	X =  351.615  mm,	Y =   -114.701  mm,	Z =   -236.484  mm,
	W =  90.000 deg,	P =   0.000 deg,	R =   90.000 deg
};
P[3234]{
   GP1:
	UF : 0, UT : 6,		CONFIG : 'N U T, 0, 0, 0',
	X =  350.642  mm,	Y =   -113.945  mm,	Z =   -236.457  mm,
	W =  90.000 deg,	P =   0.000 deg,	R =   90.000 deg
};
P[3235]{
   GP1:
	UF : 0, UT : 6,		CONFIG : 'N U T, 0, 0, 0',
	X =  349.632  mm,	Y =   -113.307  mm,	Z =   -236.452  mm,
	W =  90.000 deg,	P =   0.000 deg,	R =   90.000 deg
};
P[3236]{
   GP1:
	UF : 0, UT : 6,		CONFIG : 'N U T, 0, 0, 0',
	X =  344.937  mm,	Y =   -111.604  mm,	Z =   -236.287  mm,
	W =  90.000 deg,	P =   0.000 deg,	R =   90.000 deg
};
P[3237]{
   GP1:
	UF : 0, UT : 6,		CONFIG : 'N U T, 0, 0, 0',
	X =  342.838  mm,	Y =   -111.355  mm,	Z =   -236.028  mm,
	W =  90.000 deg,	P =   0.000 deg,	R =   90.000 deg
};
P[3238]{
   GP1:
	UF : 0, UT : 6,		CONFIG : 'N U T, 0, 0, 0',
	X =  340.930  mm,	Y =   -111.626  mm,	Z =   -236.285  mm,
	W =  90.000 deg,	P =   0.000 deg,	R =   90.000 deg
};
P[3239]{
   GP1:
	UF : 0, UT : 6,		CONFIG : 'N U T, 0, 0, 0',
	X =  338.780  mm,	Y =   -112.047  mm,	Z =   -236.080  mm,
	W =  90.000 deg,	P =   0.000 deg,	R =   90.000 deg
};
P[3240]{
   GP1:
	UF : 0, UT : 6,		CONFIG : 'N U T, 0, 0, 0',
	X =  338.192  mm,	Y =   -112.362  mm,	Z =   -236.275  mm,
	W =  90.000 deg,	P =   0.000 deg,	R =   90.000 deg
};
P[3241]{
   GP1:
	UF : 0, UT : 6,		CONFIG : 'N U T, 0, 0, 0',
	X =  337.107  mm,	Y =   -112.912  mm,	Z =   -236.405  mm,
	W =  90.000 deg,	P =   0.000 deg,	R =   90.000 deg
};
P[3242]{
   GP1:
	UF : 0, UT : 6,		CONFIG : 'N U T, 0, 0, 0',
	X =  334.503  mm,	Y =   -114.254  mm,	Z =   -236.336  mm,
	W =  90.000 deg,	P =   0.000 deg,	R =   90.000 deg
};
P[3243]{
   GP1:
	UF : 0, UT : 6,		CONFIG : 'N U T, 0, 0, 0',
	X =  331.830  mm,	Y =   -115.833  mm,	Z =   -236.422  mm,
	W =  90.000 deg,	P =   0.000 deg,	R =   90.000 deg
};
P[3244]{
   GP1:
	UF : 0, UT : 6,		CONFIG : 'N U T, 0, 0, 0',
	X =  330.177  mm,	Y =   -116.811  mm,	Z =   -236.480  mm,
	W =  90.000 deg,	P =   0.000 deg,	R =   90.000 deg
};
P[3245]{
   GP1:
	UF : 0, UT : 6,		CONFIG : 'N U T, 0, 0, 0',
	X =  327.562  mm,	Y =   -118.180  mm,	Z =   -236.136  mm,
	W =  90.000 deg,	P =   0.000 deg,	R =   90.000 deg
};
P[3246]{
   GP1:
	UF : 0, UT : 6,		CONFIG : 'N U T, 0, 0, 0',
	X =  322.354  mm,	Y =   -121.298  mm,	Z =   -236.409  mm,
	W =  90.000 deg,	P =   0.000 deg,	R =   90.000 deg
};
P[3247]{
   GP1:
	UF : 0, UT : 6,		CONFIG : 'N U T, 0, 0, 0',
	X =  321.571  mm,	Y =   -121.625  mm,	Z =   -236.103  mm,
	W =  90.000 deg,	P =   0.000 deg,	R =   90.000 deg
};
P[3248]{
   GP1:
	UF : 0, UT : 6,		CONFIG : 'N U T, 0, 0, 0',
	X =  320.626  mm,	Y =   -122.310  mm,	Z =   -236.441  mm,
	W =  90.000 deg,	P =   0.000 deg,	R =   90.000 deg
};
P[3249]{
   GP1:
	UF : 0, UT : 6,		CONFIG : 'N U T, 0, 0, 0',
	X =  319.747  mm,	Y =   -122.679  mm,	Z =   -236.108  mm,
	W =  90.000 deg,	P =   0.000 deg,	R =   90.000 deg
};
P[3250]{
   GP1:
	UF : 0, UT : 6,		CONFIG : 'N U T, 0, 0, 0',
	X =  317.760  mm,	Y =   -123.868  mm,	Z =   -236.208  mm,
	W =  90.000 deg,	P =   0.000 deg,	R =   90.000 deg
};
P[3251]{
   GP1:
	UF : 0, UT : 6,		CONFIG : 'N U T, 0, 0, 0',
	X =  317.024  mm,	Y =   -124.291  mm,	Z =   -236.201  mm,
	W =  90.000 deg,	P =   0.000 deg,	R =   90.000 deg
};
P[3252]{
   GP1:
	UF : 0, UT : 6,		CONFIG : 'N U T, 0, 0, 0',
	X =  311.457  mm,	Y =   -127.567  mm,	Z =   -236.352  mm,
	W =  90.000 deg,	P =   0.000 deg,	R =   90.000 deg
};
P[3253]{
   GP1:
	UF : 0, UT : 6,		CONFIG : 'N U T, 0, 0, 0',
	X =  308.513  mm,	Y =   -129.171  mm,	Z =   -236.117  mm,
	W =  90.000 deg,	P =   0.000 deg,	R =   90.000 deg
};
P[3254]{
   GP1:
	UF : 0, UT : 6,		CONFIG : 'N U T, 0, 0, 0',
	X =  303.378  mm,	Y =   -132.275  mm,	Z =   -236.456  mm,
	W =  90.000 deg,	P =   0.000 deg,	R =   90.000 deg
};
P[3255]{
   GP1:
	UF : 0, UT : 6,		CONFIG : 'N U T, 0, 0, 0',
	X =  302.185  mm,	Y =   -132.859  mm,	Z =   -236.203  mm,
	W =  90.000 deg,	P =   0.000 deg,	R =   90.000 deg
};
P[3256]{
   GP1:
	UF : 0, UT : 6,		CONFIG : 'N U T, 0, 0, 0',
	X =  301.114  mm,	Y =   -133.543  mm,	Z =   -236.361  mm,
	W =  90.000 deg,	P =   0.000 deg,	R =   90.000 deg
};
P[3257]{
   GP1:
	UF : 0, UT : 6,		CONFIG : 'N U T, 0, 0, 0',
	X =  299.155  mm,	Y =   -134.553  mm,	Z =   -236.068  mm,
	W =  90.000 deg,	P =   0.000 deg,	R =   90.000 deg
};
P[3258]{
   GP1:
	UF : 0, UT : 6,		CONFIG : 'N U T, 0, 0, 0',
	X =  298.148  mm,	Y =   -135.225  mm,	Z =   -236.288  mm,
	W =  90.000 deg,	P =   0.000 deg,	R =   90.000 deg
};
P[3259]{
   GP1:
	UF : 0, UT : 6,		CONFIG : 'N U T, 0, 0, 0',
	X =  295.503  mm,	Y =   -136.793  mm,	Z =   -236.386  mm,
	W =  90.000 deg,	P =   0.000 deg,	R =   90.000 deg
};
P[3260]{
   GP1:
	UF : 0, UT : 6,		CONFIG : 'N U T, 0, 0, 0',
	X =  294.548  mm,	Y =   -137.306  mm,	Z =   -236.294  mm,
	W =  90.000 deg,	P =   0.000 deg,	R =   90.000 deg
};
P[3261]{
   GP1:
	UF : 0, UT : 6,		CONFIG : 'N U T, 0, 0, 0',
	X =  291.446  mm,	Y =   -139.089  mm,	Z =   -236.273  mm,
	W =  90.000 deg,	P =   0.000 deg,	R =   90.000 deg
};
P[3262]{
   GP1:
	UF : 0, UT : 6,		CONFIG : 'N U T, 0, 0, 0',
	X =  288.476  mm,	Y =   -140.784  mm,	Z =   -236.224  mm,
	W =  90.000 deg,	P =   0.000 deg,	R =   90.000 deg
};
P[3263]{
   GP1:
	UF : 0, UT : 6,		CONFIG : 'N U T, 0, 0, 0',
	X =  287.259  mm,	Y =   -141.421  mm,	Z =   -236.065  mm,
	W =  90.000 deg,	P =   0.000 deg,	R =   90.000 deg
};
P[3264]{
   GP1:
	UF : 0, UT : 6,		CONFIG : 'N U T, 0, 0, 0',
	X =  286.391  mm,	Y =   -142.018  mm,	Z =   -236.300  mm,
	W =  90.000 deg,	P =   0.000 deg,	R =   90.000 deg
};
P[3265]{
   GP1:
	UF : 0, UT : 6,		CONFIG : 'N U T, 0, 0, 0',
	X =  283.634  mm,	Y =   -143.624  mm,	Z =   -236.331  mm,
	W =  90.000 deg,	P =   0.000 deg,	R =   90.000 deg
};
P[3266]{
   GP1:
	UF : 0, UT : 6,		CONFIG : 'N U T, 0, 0, 0',
	X =  282.240  mm,	Y =   -144.333  mm,	Z =   -236.101  mm,
	W =  90.000 deg,	P =   0.000 deg,	R =   90.000 deg
};
P[3267]{
   GP1:
	UF : 0, UT : 6,		CONFIG : 'N U T, 0, 0, 0',
	X =  280.855  mm,	Y =   -145.282  mm,	Z =   -236.463  mm,
	W =  90.000 deg,	P =   0.000 deg,	R =   90.000 deg
};
P[3268]{
   GP1:
	UF : 0, UT : 6,		CONFIG : 'N U T, 0, 0, 0',
	X =  280.155  mm,	Y =   -145.620  mm,	Z =   -236.300  mm,
	W =  90.000 deg,	P =   0.000 deg,	R =   90.000 deg
};
P[3269]{
   GP1:
	UF : 0, UT : 6,		CONFIG : 'N U T, 0, 0, 0',
	X =  279.447  mm,	Y =   -146.014  mm,	Z =   -236.266  mm,
	W =  90.000 deg,	P =   0.000 deg,	R =   90.000 deg
};
P[3270]{
   GP1:
	UF : 0, UT : 6,		CONFIG : 'N U T, 0, 0, 0',
	X =  278.600  mm,	Y =   -146.593  mm,	Z =   -236.484  mm,
	W =  90.000 deg,	P =   0.000 deg,	R =   90.000 deg
};
P[3271]{
   GP1:
	UF : 0, UT : 6,		CONFIG : 'N U T, 0, 0, 0',
	X =  276.360  mm,	Y =   -147.706  mm,	Z =   -236.045  mm,
	W =  90.000 deg,	P =   0.000 deg,	R =   90.000 deg
};
P[3272]{
   GP1:
	UF : 0, UT : 6,		CONFIG : 'N U T, 0, 0, 0',
	X =  274.173  mm,	Y =   -149.076  mm,	Z =   -236.307  mm,
	W =  90.000 deg,	P =   0.000 deg,	R =   90.000 deg
};
P[3273]{
   GP1:
	UF : 0, UT : 6,		CONFIG : 'N U T, 0, 0, 0',
	X =  272.782  mm,	Y =   -149.866  mm,	Z =   -236.275  mm,
	W =  90.000 deg,	P =   0.000 deg,	R =   90.000 deg
};
P[3274]{
   GP1:
	UF : 0, UT : 6,		CONFIG : 'N U T, 0, 0, 0',
	X =  270.771  mm,	Y =   -151.071  mm,	Z =   -236.381  mm,
	W =  90.000 deg,	P =   0.000 deg,	R =   90.000 deg
};
P[3275]{
   GP1:
	UF : 0, UT : 6,		CONFIG : 'N U T, 0, 0, 0',
	X =  268.058  mm,	Y =   -152.627  mm,	Z =   -236.356  mm,
	W =  90.000 deg,	P =   0.000 deg,	R =   90.000 deg
};
P[3276]{
   GP1:
	UF : 0, UT : 6,		CONFIG : 'N U T, 0, 0, 0',
	X =  267.254  mm,	Y =   -153.089  mm,	Z =   -236.350  mm,
	W =  90.000 deg,	P =   0.000 deg,	R =   90.000 deg
};
P[3277]{
   GP1:
	UF : 0, UT : 6,		CONFIG : 'N U T, 0, 0, 0',
	X =  264.242  mm,	Y =   -154.866  mm,	Z =   -236.442  mm,
	W =  90.000 deg,	P =   0.000 deg,	R =   90.000 deg
};
P[3278]{
   GP1:
	UF : 0, UT : 6,		CONFIG : 'N U T, 0, 0, 0',
	X =  262.448  mm,	Y =   -155.879  mm,	Z =   -236.386  mm,
	W =  90.000 deg,	P =   0.000 deg,	R =   90.000 deg
};
P[3279]{
   GP1:
	UF : 0, UT : 6,		CONFIG : 'N U T, 0, 0, 0',
	X =  261.850  mm,	Y =   -156.103  mm,	Z =   -236.091  mm,
	W =  90.000 deg,	P =   0.000 deg,	R =   90.000 deg
};
P[3280]{
   GP1:
	UF : 0, UT : 6,		CONFIG : 'N U T, 0, 0, 0',
	X =  260.892  mm,	Y =   -156.675  mm,	Z =   -236.138  mm,
	W =  90.000 deg,	P =   0.000 deg,	R =   90.000 deg
};
P[3281]{
   GP1:
	UF : 0, UT : 6,		CONFIG : 'N U T, 0, 0, 0',
	X =  257.785  mm,	Y =   -158.489  mm,	Z =   -236.187  mm,
	W =  90.000 deg,	P =   0.000 deg,	R =   90.000 deg
};
P[3282]{
   GP1:
	UF : 0, UT : 6,		CONFIG : 'N U T, 0, 0, 0',
	X =  255.250  mm,	Y =   -159.968  mm,	Z =   -236.224  mm,
	W =  90.000 deg,	P =   0.000 deg,	R =   90.000 deg
};
P[3283]{
   GP1:
	UF : 0, UT : 6,		CONFIG : 'N U T, 0, 0, 0',
	X =  252.856  mm,	Y =   -161.325  mm,	Z =   -236.164  mm,
	W =  90.000 deg,	P =   0.000 deg,	R =   90.000 deg
};
P[3284]{
   GP1:
	UF : 0, UT : 6,		CONFIG : 'N U T, 0, 0, 0',
	X =  251.892  mm,	Y =   -161.881  mm,	Z =   -236.161  mm,
	W =  90.000 deg,	P =   0.000 deg,	R =   90.000 deg
};
P[3285]{
   GP1:
	UF : 0, UT : 6,		CONFIG : 'N U T, 0, 0, 0',
	X =  250.651  mm,	Y =   -162.610  mm,	Z =   -236.192  mm,
	W =  90.000 deg,	P =   0.000 deg,	R =   90.000 deg
};
P[3286]{
   GP1:
	UF : 0, UT : 6,		CONFIG : 'N U T, 0, 0, 0',
	X =  247.122  mm,	Y =   -164.745  mm,	Z =   -236.428  mm,
	W =  90.000 deg,	P =   0.000 deg,	R =   90.000 deg
};
P[3287]{
   GP1:
	UF : 0, UT : 6,		CONFIG : 'N U T, 0, 0, 0',
	X =  242.854  mm,	Y =   -167.149  mm,	Z =   -236.281  mm,
	W =  90.000 deg,	P =   0.000 deg,	R =   90.000 deg
};
P[3288]{
   GP1:
	UF : 0, UT : 6,		CONFIG : 'N U T, 0, 0, 0',
	X =  241.892  mm,	Y =   -167.728  mm,	Z =   -236.340  mm,
	W =  90.000 deg,	P =   0.000 deg,	R =   90.000 deg
};
P[3289]{
   GP1:
	UF : 0, UT : 6,		CONFIG : 'N U T, 0, 0, 0',
	X =  241.166  mm,	Y =   -168.205  mm,	Z =   -236.481  mm,
	W =  90.000 deg,	P =   0.000 deg,	R =   90.000 deg
};
P[3290]{
   GP1:
	UF : 0, UT : 6,		CONFIG : 'N U T, 0, 0, 0',
	X =  236.767  mm,	Y =   -170.749  mm,	Z =   -236.492  mm,
	W =  90.000 deg,	P =   0.000 deg,	R =   90.000 deg
};
P[3291]{
   GP1:
	UF : 0, UT : 6,		CONFIG : 'N U T, 0, 0, 0',
	X =  234.950  mm,	Y =   -171.758  mm,	Z =   -236.391  mm,
	W =  90.000 deg,	P =   0.000 deg,	R =   90.000 deg
};
P[3292]{
   GP1:
	UF : 0, UT : 6,		CONFIG : 'N U T, 0, 0, 0',
	X =  233.916  mm,	Y =   -172.229  mm,	Z =   -236.087  mm,
	W =  90.000 deg,	P =   0.000 deg,	R =   90.000 deg
};
P[3293]{
   GP1:
	UF : 0, UT : 6,		CONFIG : 'N U T, 0, 0, 0',
	X =  229.453  mm,	Y =   -174.858  mm,	Z =   -236.213  mm,
	W =  90.000 deg,	P =   0.000 deg,	R =   90.000 deg
};
P[3294]{
   GP1:
	UF : 0, UT : 6,		CONFIG : 'N U T, 0, 0, 0',
	X =  226.068  mm,	Y =   -176.906  mm,	Z =   -236.440  mm,
	W =  90.000 deg,	P =   0.000 deg,	R =   90.000 deg
};
P[3295]{
   GP1:
	UF : 0, UT : 6,		CONFIG : 'N U T, 0, 0, 0',
	X =  224.719  mm,	Y =   -177.513  mm,	Z =   -236.022  mm,
	W =  90.000 deg,	P =   0.000 deg,	R =   90.000 deg
};
P[3296]{
   GP1:
	UF : 0, UT : 6,		CONFIG : 'N U T, 0, 0, 0',
	X =  219.349  mm,	Y =   -180.704  mm,	Z =   -236.240  mm,
	W =  90.000 deg,	P =   0.000 deg,	R =   90.000 deg
};
P[3297]{
   GP1:
	UF : 0, UT : 6,		CONFIG : 'N U T, 0, 0, 0',
	X =  215.397  mm,	Y =   -183.015  mm,	Z =   -236.313  mm,
	W =  90.000 deg,	P =   0.000 deg,	R =   90.000 deg
};
P[3298]{
   GP1:
	UF : 0, UT : 6,		CONFIG : 'N U T, 0, 0, 0',
	X =  214.049  mm,	Y =   -183.679  mm,	Z =   -236.034  mm,
	W =  90.000 deg,	P =   0.000 deg,	R =   90.000 deg
};
P[3299]{
   GP1:
	UF : 0, UT : 6,		CONFIG : 'N U T, 0, 0, 0',
	X =  211.182  mm,	Y =   -185.383  mm,	Z =   -236.153  mm,
	W =  90.000 deg,	P =   0.000 deg,	R =   90.000 deg
};
P[3300]{
   GP1:
	UF : 0, UT : 6,		CONFIG : 'N U T, 0, 0, 0',
	X =  207.300  mm,	Y =   -187.731  mm,	Z =   -236.410  mm,
	W =  90.000 deg,	P =   0.000 deg,	R =   90.000 deg
};
P[3301]{
   GP1:
	UF : 0, UT : 6,		CONFIG : 'N U T, 0, 0, 0',
	X =  205.364  mm,	Y =   -188.720  mm,	Z =   -236.098  mm,
	W =  90.000 deg,	P =   0.000 deg,	R =   90.000 deg
};
P[3302]{
   GP1:
	UF : 0, UT : 6,		CONFIG : 'N U T, 0, 0, 0',
	X =  203.957  mm,	Y =   -189.647  mm,	Z =   -236.377  mm,
	W =  90.000 deg,	P =   0.000 deg,	R =   90.000 deg
};
P[3303]{
   GP1:
	UF : 0, UT : 6,		CONFIG : 'N U T, 0, 0, 0',
	X =  199.839  mm,	Y =   -191.990  mm,	Z =   -236.293  mm,
	W =  90.000 deg,	P =   0.000 deg,	R =   90.000 deg
};
P[3304]{
   GP1:
	UF : 0, UT : 6,		CONFIG : 'N U T, 0, 0, 0',
	X =  198.334  mm,	Y =   -192.757  mm,	Z =   -236.045  mm,
	W =  90.000 deg,	P =   0.000 deg,	R =   90.000 deg
};
P[3305]{
   GP1:
	UF : 0, UT : 6,		CONFIG : 'N U T, 0, 0, 0',
	X =  194.437  mm,	Y =   -195.137  mm,	Z =   -236.362  mm,
	W =  90.000 deg,	P =   0.000 deg,	R =   90.000 deg
};
P[3306]{
   GP1:
	UF : 0, UT : 6,		CONFIG : 'N U T, 0, 0, 0',
	X =  190.579  mm,	Y =   -197.285  mm,	Z =   -236.166  mm,
	W =  90.000 deg,	P =   0.000 deg,	R =   90.000 deg
};
P[3307]{
   GP1:
	UF : 0, UT : 6,		CONFIG : 'N U T, 0, 0, 0',
	X =  189.500  mm,	Y =   -198.043  mm,	Z =   -236.494  mm,
	W =  90.000 deg,	P =   0.000 deg,	R =   90.000 deg
};
P[3308]{
   GP1:
	UF : 0, UT : 6,		CONFIG : 'N U T, 0, 0, 0',
	X =  188.455  mm,	Y =   -198.573  mm,	Z =   -236.316  mm,
	W =  90.000 deg,	P =   0.000 deg,	R =   90.000 deg
};
P[3309]{
   GP1:
	UF : 0, UT : 6,		CONFIG : 'N U T, 0, 0, 0',
	X =  187.079  mm,	Y =   -199.250  mm,	Z =   -236.032  mm,
	W =  90.000 deg,	P =   0.000 deg,	R =   90.000 deg
};
P[3310]{
   GP1:
	UF : 0, UT : 6,		CONFIG : 'N U T, 0, 0, 0',
	X =  184.549  mm,	Y =   -200.840  mm,	Z =   -236.344  mm,
	W =  90.000 deg,	P =   0.000 deg,	R =   90.000 deg
};
P[3311]{
   GP1:
	UF : 0, UT : 6,		CONFIG : 'N U T, 0, 0, 0',
	X =  182.860  mm,	Y =   -201.804  mm,	Z =   -236.317  mm,
	W =  90.000 deg,	P =   0.000 deg,	R =   90.000 deg
};
P[3312]{
   GP1:
	UF : 0, UT : 6,		CONFIG : 'N U T, 0, 0, 0',
	X =  181.154  mm,	Y =   -202.750  mm,	Z =   -236.223  mm,
	W =  90.000 deg,	P =   0.000 deg,	R =   90.000 deg
};
P[3313]{
   GP1:
	UF : 0, UT : 6,		CONFIG : 'N U T, 0, 0, 0',
	X =  178.452  mm,	Y =   -204.373  mm,	Z =   -236.377  mm,
	W =  90.000 deg,	P =   0.000 deg,	R =   90.000 deg
};
P[3314]{
   GP1:
	UF : 0, UT : 6,		CONFIG : 'N U T, 0, 0, 0',
	X =  177.530  mm,	Y =   -204.912  mm,	Z =   -236.393  mm,
	W =  90.000 deg,	P =   0.000 deg,	R =   90.000 deg
};
P[3315]{
   GP1:
	UF : 0, UT : 6,		CONFIG : 'N U T, 0, 0, 0',
	X =  174.367  mm,	Y =   -206.663  mm,	Z =   -236.212  mm,
	W =  90.000 deg,	P =   0.000 deg,	R =   90.000 deg
};
P[3316]{
   GP1:
	UF : 0, UT : 6,		CONFIG : 'N U T, 0, 0, 0',
	X =  173.461  mm,	Y =   -207.307  mm,	Z =   -236.503  mm,
	W =  90.000 deg,	P =   0.000 deg,	R =   90.000 deg
};
P[3317]{
   GP1:
	UF : 0, UT : 6,		CONFIG : 'N U T, 0, 0, 0',
	X =  169.461  mm,	Y =   -209.616  mm,	Z =   -236.502  mm,
	W =  90.000 deg,	P =   0.000 deg,	R =   90.000 deg
};
P[3318]{
   GP1:
	UF : 0, UT : 6,		CONFIG : 'N U T, 0, 0, 0',
	X =  168.601  mm,	Y =   -210.029  mm,	Z =   -236.299  mm,
	W =  90.000 deg,	P =   0.000 deg,	R =   90.000 deg
};
P[3319]{
   GP1:
	UF : 0, UT : 6,		CONFIG : 'N U T, 0, 0, 0',
	X =  165.948  mm,	Y =   -211.632  mm,	Z =   -236.473  mm,
	W =  90.000 deg,	P =   0.000 deg,	R =   90.000 deg
};
P[3320]{
   GP1:
	UF : 0, UT : 6,		CONFIG : 'N U T, 0, 0, 0',
	X =  164.809  mm,	Y =   -212.300  mm,	Z =   -236.496  mm,
	W =  90.000 deg,	P =   0.000 deg,	R =   90.000 deg
};
P[3321]{
   GP1:
	UF : 0, UT : 6,		CONFIG : 'N U T, 0, 0, 0',
	X =  163.979  mm,	Y =   -212.755  mm,	Z =   -236.439  mm,
	W =  90.000 deg,	P =   0.000 deg,	R =   90.000 deg
};
P[3322]{
   GP1:
	UF : 0, UT : 6,		CONFIG : 'N U T, 0, 0, 0',
	X =  162.248  mm,	Y =   -213.708  mm,	Z =   -236.325  mm,
	W =  90.000 deg,	P =   0.000 deg,	R =   90.000 deg
};
P[3323]{
   GP1:
	UF : 0, UT : 6,		CONFIG : 'N U T, 0, 0, 0',
	X =  158.062  mm,	Y =   -216.196  mm,	Z =   -236.498  mm,
	W =  90.000 deg,	P =   0.000 deg,	R =   90.000 deg
};
P[3324]{
   GP1:
	UF : 0, UT : 6,		CONFIG : 'N U T, 0, 0, 0',
	X =  154.773  mm,	Y =   -218.093  mm,	Z =   -236.493  mm,
	W =  90.000 deg,	P =   0.000 deg,	R =   90.000 deg
};
P[3325]{
   GP1:
	UF : 0, UT : 6,		CONFIG : 'N U T, 0, 0, 0',
	X =  153.501  mm,	Y =   -218.759  mm,	Z =   -236.324  mm,
	W =  90.000 deg,	P =   0.000 deg,	R =   90.000 deg
};
P[3326]{
   GP1:
	UF : 0, UT : 6,		CONFIG : 'N U T, 0, 0, 0',
	X =  152.751  mm,	Y =   -219.156  mm,	Z =   -236.239  mm,
	W =  90.000 deg,	P =   0.000 deg,	R =   90.000 deg
};
P[3327]{
   GP1:
	UF : 0, UT : 6,		CONFIG : 'N U T, 0, 0, 0',
	X =  151.575  mm,	Y =   -219.935  mm,	Z =   -236.482  mm,
	W =  90.000 deg,	P =   0.000 deg,	R =   90.000 deg
};
P[3328]{
   GP1:
	UF : 0, UT : 6,		CONFIG : 'N U T, 0, 0, 0',
	X =  144.993  mm,	Y =   -223.722  mm,	Z =   -236.449  mm,
	W =  90.000 deg,	P =   0.000 deg,	R =   90.000 deg
};
P[3329]{
   GP1:
	UF : 0, UT : 6,		CONFIG : 'N U T, 0, 0, 0',
	X =  141.405  mm,	Y =   -225.684  mm,	Z =   -236.183  mm,
	W =  90.000 deg,	P =   0.000 deg,	R =   90.000 deg
};
P[3330]{
   GP1:
	UF : 0, UT : 6,		CONFIG : 'N U T, 0, 0, 0',
	X =  140.527  mm,	Y =   -226.243  mm,	Z =   -236.310  mm,
	W =  90.000 deg,	P =   0.000 deg,	R =   90.000 deg
};
P[3331]{
   GP1:
	UF : 0, UT : 6,		CONFIG : 'N U T, 0, 0, 0',
	X =  139.467  mm,	Y =   -226.889  mm,	Z =   -236.392  mm,
	W =  90.000 deg,	P =   0.000 deg,	R =   90.000 deg
};
P[3332]{
   GP1:
	UF : 0, UT : 6,		CONFIG : 'N U T, 0, 0, 0',
	X =  138.561  mm,	Y =   -227.345  mm,	Z =   -236.228  mm,
	W =  90.000 deg,	P =   0.000 deg,	R =   90.000 deg
};
P[3333]{
   GP1:
	UF : 0, UT : 6,		CONFIG : 'N U T, 0, 0, 0',
	X =  136.064  mm,	Y =   -228.853  mm,	Z =   -236.389  mm,
	W =  90.000 deg,	P =   0.000 deg,	R =   90.000 deg
};
P[3334]{
   GP1:
	UF : 0, UT : 6,		CONFIG : 'N U T, 0, 0, 0',
	X =  134.622  mm,	Y =   -229.718  mm,	Z =   -236.468  mm,
	W =  90.000 deg,	P =   0.000 deg,	R =   90.000 deg
};
P[3335]{
   GP1:
	UF : 0, UT : 6,		CONFIG : 'N U T, 0, 0, 0',
	X =  132.531  mm,	Y =   -230.898  mm,	Z =   -236.400  mm,
	W =  90.000 deg,	P =   0.000 deg,	R =   90.000 deg
};
P[3336]{
   GP1:
	UF : 0, UT : 6,		CONFIG : 'N U T, 0, 0, 0',
	X =  131.000  mm,	Y =   -231.707  mm,	Z =   -236.220  mm,
	W =  90.000 deg,	P =   0.000 deg,	R =   90.000 deg
};
P[3337]{
   GP1:
	UF : 0, UT : 6,		CONFIG : 'N U T, 0, 0, 0',
	X =  129.867  mm,	Y =   -232.415  mm,	Z =   -236.350  mm,
	W =  90.000 deg,	P =   0.000 deg,	R =   90.000 deg
};
P[3338]{
   GP1:
	UF : 0, UT : 6,		CONFIG : 'N U T, 0, 0, 0',
	X =  126.987  mm,	Y =   -234.098  mm,	Z =   -236.400  mm,
	W =  90.000 deg,	P =   0.000 deg,	R =   90.000 deg
};
P[3339]{
   GP1:
	UF : 0, UT : 6,		CONFIG : 'N U T, 0, 0, 0',
	X =  126.039  mm,	Y =   -234.684  mm,	Z =   -236.492  mm,
	W =  90.000 deg,	P =   0.000 deg,	R =   90.000 deg
};
P[3340]{
   GP1:
	UF : 0, UT : 6,		CONFIG : 'N U T, 0, 0, 0',
	X =  124.194  mm,	Y =   -235.553  mm,	Z =   -236.017  mm,
	W =  90.000 deg,	P =   0.000 deg,	R =   90.000 deg
};
P[3341]{
   GP1:
	UF : 0, UT : 6,		CONFIG : 'N U T, 0, 0, 0',
	X =  122.043  mm,	Y =   -236.854  mm,	Z =   -236.159  mm,
	W =  90.000 deg,	P =   0.000 deg,	R =   90.000 deg
};
P[3342]{
   GP1:
	UF : 0, UT : 6,		CONFIG : 'N U T, 0, 0, 0',
	X =  120.134  mm,	Y =   -237.930  mm,	Z =   -236.096  mm,
	W =  90.000 deg,	P =   0.000 deg,	R =   90.000 deg
};
P[3343]{
   GP1:
	UF : 0, UT : 6,		CONFIG : 'N U T, 0, 0, 0',
	X =  118.307  mm,	Y =   -239.097  mm,	Z =   -236.370  mm,
	W =  90.000 deg,	P =   0.000 deg,	R =   90.000 deg
};
P[3344]{
   GP1:
	UF : 0, UT : 6,		CONFIG : 'N U T, 0, 0, 0',
	X =  114.302  mm,	Y =   -241.469  mm,	Z =   -236.512  mm,
	W =  90.000 deg,	P =   0.000 deg,	R =   90.000 deg
};
P[3345]{
   GP1:
	UF : 0, UT : 6,		CONFIG : 'N U T, 0, 0, 0',
	X =  112.360  mm,	Y =   -242.438  mm,	Z =   -236.141  mm,
	W =  90.000 deg,	P =   0.000 deg,	R =   90.000 deg
};
P[3346]{
   GP1:
	UF : 0, UT : 6,		CONFIG : 'N U T, 0, 0, 0',
	X =  111.300  mm,	Y =   -243.144  mm,	Z =   -236.372  mm,
	W =  90.000 deg,	P =   0.000 deg,	R =   90.000 deg
};
P[3347]{
   GP1:
	UF : 0, UT : 6,		CONFIG : 'N U T, 0, 0, 0',
	X =  109.357  mm,	Y =   -244.289  mm,	Z =   -236.427  mm,
	W =  90.000 deg,	P =   0.000 deg,	R =   90.000 deg
};
P[3348]{
   GP1:
	UF : 0, UT : 6,		CONFIG : 'N U T, 0, 0, 0',
	X =  107.937  mm,	Y =   -245.015  mm,	Z =   -236.199  mm,
	W =  90.000 deg,	P =   0.000 deg,	R =   90.000 deg
};
P[3349]{
   GP1:
	UF : 0, UT : 6,		CONFIG : 'N U T, 0, 0, 0',
	X =  104.572  mm,	Y =   -247.010  mm,	Z =   -236.327  mm,
	W =  90.000 deg,	P =   0.000 deg,	R =   90.000 deg
};
P[3350]{
   GP1:
	UF : 0, UT : 6,		CONFIG : 'N U T, 0, 0, 0',
	X =  195.000  mm,	Y =   -410.000  mm,	Z =   -250.000  mm,
	W =  90.000 deg,	P =   0.000 deg,	R =   90.000 deg
};
/END
